FUNCTION_BLOCK FB_SEL_ARRAY (* ARRAY Selection *)
  (* Standard: IEC 61499; Function: Selection; Type: ARRAY *)
  (* Version 0.2, 2007-10-26, JHC, Holobloc Inc, Updated documentation. *)
  (* Version 0.1, 2006-09-13, JHC, Holobloc Inc, Moved to fb.rt.select. *)
  (* Version 0.0, 2004-12-15, JHC, Rockwell Automation, Converted from SRC format. *)
  (* Compiler header: package fb.rt.select; *)
  (* Compiler Java Sun JDK 1.6.0 *)
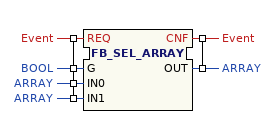
  EVENT_INPUT
    REQ WITH G, IN0, IN1;
  END_EVENT
  EVENT_OUTPUT
    CNF WITH OUT;
  END_EVENT
  VAR_INPUT
    G : BOOL; (* Selector *)
    IN0 : ARRAY; (* Selected when G=0 *)
    IN1 : ARRAY; (* Selected when G=1 *)
  END_VAR
  VAR_OUTPUT
    OUT : ARRAY; (* Selected value *)
  END_VAR
END_FUNCTION_BLOCK
